// Alarm sensor FB
FUNCTION_BLOCK FB_AlarmSensor IMPLEMENTS I_AlarmSensor
VAR
	sName					: STRING;				// Sensor name
	nID						: INT;					// Alarm component ID
	bWarnFirst				: BOOL;					// Set to true to warn the user before setting off the alarm
	
	ibAlarm			AT %I*	: BOOL;					// Active low alarm input
	ibTamper		AT %I*	: BOOL;					// Active low tamper input
	
	bAlarm					: BOOL;					// True if the sensor detects something
	bTamper					: BOOL;					// True if the sensor is tampered with
	
	bAlarmTrigger			: BOOL;					// Returns true when the sensor is triggered
	bTamperTrigger			: BOOL;					// Returns true when the sensor is tampered with
	
	stHMI					: ST_AlarmSensorHMI;	// HMI data
END_VAR

// Returns true if the sensor detects something (as long as something is detected)
PROPERTY Alarm : BOOL
GET
Alarm := bAlarm;
END_GET
END_PROPERTY

// Returns true when the sensor is triggered (one cycle)
PROPERTY AlarmTrigger : BOOL
GET
AlarmTrigger := bAlarmTrigger;
END_GET
END_PROPERTY

// Run this method every cycle
METHOD Execute
VAR_INST
	fbAlarm		: R_TRIG;		// Alarm rising trigger
	fbTamper	: R_TRIG;		// Tamper rising trigger
END_VAR
// Convert active low inputs
bAlarm := NOT ibAlarm;
bTamper := NOT ibTamper;

// Run FBs
fbAlarm(CLK := bAlarm);
fbTamper(CLK := bTamper);

// Check triggers
bAlarmTrigger := fbAlarm.Q;
bTamperTrigger := fbTamper.Q;

// Update HMI
UpdateHMI();
END_METHOD

METHOD FB_init : BOOL
VAR_INPUT
	bInitRetains	: BOOL;		// if TRUE, the retain variables are initialized (warm start / cold start)
	bInCopyCode		: BOOL;		// if TRUE, the instance afterwards gets moved into the copy code (online change)
	
	sSensorName		: STRING;	// Sensor name
	nSensorID		: INT;		// Sensor ID
	bEnableWarning	: BOOL;		// Set to true to warn the user before setting off the alarm
END_VAR
sName := sSensorName;
nID := nSensorID;
bWarnFirst := bEnableWarning;
END_METHOD

// Returns the HMI data
PROPERTY HmiData : ST_AlarmSensorHMI
GET
HmiData := stHMI;
END_GET
END_PROPERTY

// Get the alarm component ID of the sensor
PROPERTY ID : INT
GET
ID := nID;
END_GET
END_PROPERTY

// Returns true when the sensor is tampered with (as long as the sensor is tampered with)
PROPERTY Tamper : BOOL
GET
Tamper := bTamper;
END_GET
END_PROPERTY

// Returns true when the tamper sensor is triggered (one cycle)
PROPERTY TamperTrigger : BOOL
GET
TamperTrigger := bTamperTrigger;
END_GET
END_PROPERTY

// Update HMI
METHOD PRIVATE UpdateHMI
stHMI.sName := sName;
stHMI.nID := nID;
stHMI.bAlarm := bAlarm;
stHMI.bTamper := bTamper;
END_METHOD

// Returs true if the user is warned before the alarm is set off
PROPERTY WarnFirst : BOOL
GET
WarnFirst := bWarnFirst;
END_GET
END_PROPERTY

END_FUNCTION_BLOCK

(* stored: Version 1.1.0.1, ProductVersion 3.1.4024.12
   POU FB_AlarmSensor: Id {b70c0fc3-adeb-4f9c-974b-1c2e4d76696e}, SpecialFunc None
   Folder Methods: Id {51ed284b-55ce-458c-9d89-521a2a263c5a}
   Folder Properties: Id {c1a533fb-ae32-4976-947d-2ef3acce91e4}
   Property Alarm: Id {dc64478c-441d-49da-8224-efa81b6d9483}
   Get Get: Id {0272ca24-d09e-4e5b-9b48-31f9e8b81725}
   Property AlarmTrigger: Id {12666827-13e2-4f8c-9bf9-2a8a411f7a47}
   Get Get: Id {f6a62fa3-d0aa-45ff-b344-75a4803e9461}
   Method Execute: Id {0f046a5a-16a3-4b62-b056-a50c4fc1278a}
   Method FB_init: Id {ff1dc40c-1996-4aae-aa5c-8b8b146a64eb}
   Property HmiData: Id {11eea628-f2e6-4a99-a31a-35cef36b6bfd}
   Get Get: Id {62f261ad-958a-4521-9634-bca43aa5fca2}
   Property ID: Id {2b131cc5-68f4-47ea-996b-1741c668fec3}
   Get Get: Id {d94e6bc9-789d-4574-bf17-ba645a08e35a}
   Property Tamper: Id {a2a0dd8d-69b1-4bb6-a23a-ef712e963b3a}
   Get Get: Id {615b5d68-2aab-4f4c-9b3f-662b04191962}
   Property TamperTrigger: Id {eb07d766-9369-49d4-b8a5-9ec5e976e5da}
   Get Get: Id {39814ef7-3c13-42fe-a6cb-dd65a495ad1d}
   Method UpdateHMI: Id {2a73659b-cde5-47f2-97a4-eb437262e9fa}
   Property WarnFirst: Id {8b5a5135-7729-4535-8e9c-5ce7d3db4bc8}
   Get Get: Id {e88c85de-9f8d-444d-973e-afb2649b79d6} *)
